		ProdAER_1T_realtime := (INT_TO_REAL(ProducaoProgramada_AER_1T) / (MinDispAER_1T)) * ((
		(INT_TO_REAL(hora)-INT_TO_REAL(HoraInicio1Turno))*60)-INT_TO_REAL(MinInicio1Turno) + INT_TO_REAL(minuto)-10-20-15);
	
		EficAER_1T_realtime := ( INT_TO_REAL(CNT_PRD_AER_1T) / ProdAER_1T_realtime ) * 100;
		END_IF
		
				IF hora > 12 AND hora < 15 AND minuto < 9 THEN

		ProdAER_1T_realtime := (INT_TO_REAL(ProducaoProgramada_AER_1T) / (MinDispAER_1T)) * ((
		(INT_TO_REAL(hora)-INT_TO_REAL(HoraInicio1Turno))*60)-INT_TO_REAL(MinInicio1Turno) + INT_TO_REAL(minuto)-10-20-15-60-10);
	
		EficAER_1T_realtime := ( INT_TO_REAL(CNT_PRD_AER_1T) / ProdAER_1T_realtime ) * 100;
		END_IF
//HABILITA RTC==========================
	IF xEnable = TRUE THEN
	Result := GetDateAndTime(DATEANDTIME);
	END_IF
//HABILITA RTC==========================

//==============Habilita contadores 1º turno ================
IF (hora = HoraInicio1Turno AND minuto = MinInicio1Turno)  THEN
HabContAER_1T := TRUE;
HabContAER_3T := FALSE;
END_IF 


//==============Contador e Eficiencia AER 1 TURNO de cartuchos==========
IF HabContAER_1T = TRUE THEN 
PULSO_CNT_AER_1T(CLK:=CNT_AER);	
		IF PULSO_CNT_AER_1T.Q = TRUE THEN
		CNT_PRD_AER_1T := CNT_PRD_AER_1T+1;	
		END_IF
END_IF
EficienciaAER_1T := (INT_TO_REAL(CNT_PRD_AER_1T) / INT_TO_REAL(ProducaoProgramada_AER_1T) ) * 100;

//=====================1º TURNO ========================

//=====================2º TURNO ========================

	//10 minutos - Reunião / DSS / Treinamento
	//20 minutosPartida de linha / Parada de Linha
	//15 minutosRefeições (Café / Almoço / Janta)
	//60 minutosRefeições (Café / Almoço / Janta)
	//10 minutosPartida de linha / Parada de Linha
	IF hora = 0 THEN 
		hora := 24;
	END_IF
	
		MinDispAER_2T := (((INT_TO_REAL (HoraFim2Turno) - INT_TO_REAL(HoraInicio2Turno) )*60)-
		INT_TO_REAL(MinInicio2Turno)+INT_TO_REAL(MinFim2Turno)-10-20-15-60-10);
		
	IF (hora > 15 AND minuto > 8) AND hora < 17 THEN

		ProdAER_2T_realtime := (INT_TO_REAL(ProducaoProgramada_AER_2T) / (MinDispAER_2T)) * ((
		(INT_TO_REAL(hora)-INT_TO_REAL(HoraInicio2Turno))*60)-INT_TO_REAL(MinInicio2Turno) + INT_TO_REAL(minuto)-10-20);
	
		EficAER_2T_realtime := ( INT_TO_REAL(CNT_PRD_AER_2T) / ProdAER_2T_realtime ) * 100;
		END_IF
		
			IF hora > 17 AND hora < 20 THEN

		ProdAER_2T_realtime := (INT_TO_REAL(ProducaoProgramada_AER_2T) / (MinDispAER_2T)) * ((
		(INT_TO_REAL(hora)-INT_TO_REAL(HoraInicio2Turno))*60)-INT_TO_REAL(MinInicio2Turno) + INT_TO_REAL(minuto)-10-20-15);
	
		EficAER_2T_realtime := ( INT_TO_REAL(CNT_PRD_AER_2T) / ProdAER_2T_realtime ) * 100;
		END_IF
		
				IF hora > 20 AND hora < 24 THEN

		ProdAER_2T_realtime := (INT_TO_REAL(ProducaoProgramada_AER_2T) / (MinDispAER_2T)) * ((
		(INT_TO_REAL(hora)-INT_TO_REAL(HoraInicio2Turno))*60)-INT_TO_REAL(MinInicio2Turno) + INT_TO_REAL(minuto)-10-20-15-60-10);
	
		EficAER_2T_realtime := ( INT_TO_REAL(CNT_PRD_AER_2T) / ProdAER_2T_realtime ) * 100;
		END_IF
//==============Contador e Eficiencia AER 2 TURNO de cartuchos==========
//==============Habilita contadores 2º turno ================
IF (hora = HoraInicio2Turno AND minuto = MinInicio2Turno)  THEN
HabContAER_2T := TRUE;
HabContAER_1T := FALSE;
END_IF 
IF HabContAER_2T = TRUE THEN 
PULSO_CNT_AER_2T(CLK:=CNT_AER);	
		IF PULSO_CNT_AER_2T.Q = TRUE THEN
		CNT_PRD_AER_2T := CNT_PRD_AER_2T+1;	
		END_IF
END_IF
EficienciaAER_2T := (INT_TO_REAL (CNT_PRD_AER_2T) / INT_TO_REAL (ProducaoProgramada_AER_2T)  ) * 100;

//=====================2º TURNO ========================

//=====================3º TURNO ========================
//==============Contador e Eficiencia AER 3 TURNO de cartuchos==========

//==============Habilita contadores 3º turno ================
//10 minutos - Reunião / DSS / Treinamento
	//20 minutosPartida de linha / Parada de Linha
	//15 minutosRefeições (Café / Almoço / Janta)
	//60 minutosRefeições (Café / Almoço / Janta)
	//10 minutosPartida de linha / Parada de Linha
	IF hora = 0 THEN 
		hora := 24;
	END_IF
	
		MinDispAER_3T := (((INT_TO_REAL (HoraFim3Turno) - INT_TO_REAL(HoraInicio3Turno) )*60)-
		INT_TO_REAL(MinInicio3Turno)+INT_TO_REAL(MinFim3Turno)-10-20-15-60-10);
		
	IF ((hora > 0 OR hora = 24) AND minuto > 32) AND hora < 02 THEN

		ProdAER_3T_realtime := (INT_TO_REAL(ProducaoProgramada_AER_3T) / (MinDispAER_3T)) * ((
		(INT_TO_REAL(hora)-INT_TO_REAL(HoraInicio3Turno))*60)-INT_TO_REAL(MinInicio3Turno) + INT_TO_REAL(minuto)-10-20);
	
		EficAER_3T_realtime := ( INT_TO_REAL(CNT_PRD_AER_3T) / ProdAER_3T_realtime ) * 100;
		END_IF
		
			IF hora > 17 AND hora < 20 THEN

		ProdAER_3T_realtime := (INT_TO_REAL(ProducaoProgramada_AER_3T) / (MinDispAER_3T)) * ((
		(INT_TO_REAL(hora)-INT_TO_REAL(HoraInicio3Turno))*60)-INT_TO_REAL(MinInicio3Turno) + INT_TO_REAL(minuto)-10-20-15);
	
		EficAER_3T_realtime := ( INT_TO_REAL(CNT_PRD_AER_3T) / ProdAER_3T_realtime ) * 100;
		END_IF
		
				IF hora > 20 AND hora < 24 THEN

		ProdAER_3T_realtime := (INT_TO_REAL(ProducaoProgramada_AER_3T) / (MinDispAER_3T)) * ((
		(INT_TO_REAL(hora)-INT_TO_REAL(HoraInicio3Turno))*60)-INT_TO_REAL(MinInicio3Turno) + INT_TO_REAL(minuto)-10-20-15-60-10);
	
		EficAER_3T_realtime := ( INT_TO_REAL(CNT_PRD_AER_3T) / ProdAER_3T_realtime ) * 100;
		END_IF
//==============Contador e Eficiencia AER 3 TURNO de cartuchos==========
//==============Habilita contadores 3º turno ================
IF (hora = HoraInicio3Turno AND minuto = MinInicio3Turno)  THEN
HabContAER_3T := TRUE;
HabContAER_2T := FALSE;
END_IF 
IF HabContAER_3T = TRUE THEN 
PULSO_CNT_AER_3T(CLK:=CNT_AER);	
		IF PULSO_CNT_AER_3T.Q = TRUE THEN
		CNT_PRD_AER_3T := CNT_PRD_AER_3T+1;	
		END_IF
END_IF
EficienciaAER_3T := (INT_TO_REAL (CNT_PRD_AER_3T) / INT_TO_REAL (ProducaoProgramada_AER_3T)  ) * 100;


IF (hora = HoraInicio3Turno AND minuto = MinInicio3Turno)  THEN
HabContAER_3T := TRUE;
HabContAER_2T := FALSE;
END_IF 
IF HabContAER_3T = TRUE THEN 
PULSO_CNT_AER_3T(CLK:=CNT_AER);	
		IF PULSO_CNT_AER_3T.Q = TRUE THEN
		CNT_PRD_AER_3T := CNT_PRD_AER_3T+1;	
		END_IF
END_IF
EficienciaAER_3T := (INT_TO_REAL (CNT_PRD_AER_3T) / INT_TO_REAL(ProducaoProgramada_AER_3T)  ) * 100;
//=====================3º TURNO ========================

END_PROGRAM

// Device/Application/ampliacao_transferencia
PROGRAM ampliacao_transferencia

VAR
	BA_03_INV : INV_MODBUS;
	BB_02_INV : INV_MODBUS;
	MH_01_INV : INV_MODBUS;
	MH_02_INV : INV_MODBUS;
	
	AUX_BA_03_HAB : BOOL;
	AUX_BB_02_HAB : BOOL;
	AUX_MH_01_HAB : BOOL;
	AUX_MH_02_HAB : BOOL;
	AUX_BA_03_PRESET: REAL;
	CTRL_BB2 : PD;
	BB_02_PRT_MAN : BOOL;
	AUX_BA_03_FLT_PRESS : BOOL;
	
	AUX_BB2_PRST_VEL : REAL;
	
	
	R_BB_02_REF_VEL : REAL;
	R_PRST_PRESS_BB : REAL;
	R_BB_02_PRS_VEL : REAL;
	
	
	TMR_FALHA_PRESSAO_BBALTA3_ALARME : TON;
END_VAR


(* PARAMENTROS DO INVERSOR DA BOMBA DE ALTA PRESSÃO 03*)
BA_03_INV (
	LIGA := BA_03_CMDS,
	CMD_RESET := BTS_RSTAL,
	CMD_STOP := AL_GERAL,
	CMD_HAB := AUX_BA_03_HAB,
	REF_VEL := BA_03_REF_VEL,
	STATUS := BA_03_ST,
	FALHA := BA_03_FLT,
	PRESET := AUX_BA_03_PRESET,
	LIGADO => BA_03_CMD,
	HABILITADO => BA_03_HAB,
	STOP => BA_03_STP,
	RESET => BA_03_RST,
	VEL => BA_03_ST_VELS,
	STS_INV => BA_03_STS,
	FLT_INV => BA_03_FLTS,
	PRT_VEL => BA_03_PRS_VEL);
	
	
	(* PARAMENTROS DO INVERSOR DA BOMBA DE BAIXA PRESSÃO 02*)
BB_02_INV (
	LIGA := BB_02_CMDS,
	CMD_RESET := BTS_RSTAL,
	CMD_STOP := AL_GERAL,
	CMD_HAB := AUX_BB_02_HAB,
	//REF_VEL := 
	STATUS := BB_02_ST,
	FALHA := BB_02_FLT,
	PRESET := AUX_BB2_PRST_VEL,
	LIGADO => BB_02_CMD,
	HABILITADO => BB_02_HAB,
	STOP => BB_02_STP,
	RESET => BB_02_RST,
	//VEL => 
	STS_INV => BB_02_STS,
	FLT_INV => BB_02_FLTS,
	PRT_VEL => BB_02_PRS_VEL);
	
		(* PARAMENTROS DO INVERSOR DO MOINHO 01*)
MH_01_INV (
	LIGA := MH_01_CMDS,
	CMD_RESET := BTS_RSTAL,
	CMD_STOP := AL_GERAL,
	CMD_HAB := AUX_MH_01_HAB,
	//REF_VEL := 
	STATUS := MH_01_ST,
	FALHA := MH_01_FLT,
	//PRESET := 
	LIGADO => MH_01_CMD,
	HABILITADO => MH_01_HAB,
	STOP => MH_01_STP,
	RESET => MH_01_RST,
	//VEL => 
	STS_INV => MH_01_STS,
	FLT_INV => MH_01_FLTS,
	//PRT_VEL => 
);

	(* PARAMENTROS DO INVERSOR DO MOINHO 01*)
MH_02_INV (
	LIGA := MH_02_CMDS,
	CMD_RESET := BTS_RSTAL,
	CMD_STOP := AL_GERAL,
	CMD_HAB := AUX_MH_02_HAB,
	//REF_VEL := 
	STATUS := MH_02_ST,
	FALHA := MH_02_FLT,
	//PRESET := 
	LIGADO => MH_02_CMD,
	HABILITADO => MH_02_HAB,
	STOP => MH_02_STP,
	RESET => MH_02_RST,
	//VEL => 
	STS_INV => MH_02_STS,
	FLT_INV => MH_02_FLTS,
	//PRT_VEL => 
);

                   (*LOGICA DA BOMBA DE ALTA 03*)
//----------------------------------------------------------------------------------

//COMANDO LIGA DA BOMBA DE ALTA 03				   
IF  (SD_BB=TRUE OR BB_02_ST = TRUE) AND  PRESSAO_ALTA_LINHA_ALTA = FALSE THEN
IF (NOT SD_BA1) OR (NOT SD_BA2) THEN
	AUX_BA_03_HAB := TRUE;
	END_IF
END_IF

//SETPOINT VELOCIDADE DE BOMBA DE ALTA 03
IF BA_03_ST THEN
	AUX_BA_03_PRESET := PRST_VEL_BA1;
	ELSE 
		AUX_BA_03_PRESET := 0;
	END_IF

                   (*LOGICA DA BOMBA DE BAIXA 02*)
//----------------------------------------------------------------------------------

// COMANDO LLIGA DA BOMBA DE BAIXA 02
	IF SD_BB = FALSE AND NIVEL_MINIMO_MXE = FALSE AND PRESSAO_ALTA_LINHA_ALTA = FALSE THEN
	AUX_BB_02_HAB := TRUE;
	ELSE
	AUX_BB_02_HAB := FALSE;
END_IF
	//move velocidade da bomba de baixa 02 em manual
 IF (BB_02_ST = TRUE AND BB_AUTOM = FALSE) THEN
		AUX_BB2_PRST_VEL := BB_02_PRS_VEL;
	
END_IF
		
	
	// SETPIOINT VAI A ZERO SE NAO ESTIVER FUNCIONANDO
IF BB_02_ST = FALSE THEN 
	AUX_BB2_PRST_VEL := 0;
	END_IF
	
		//move velocidade da bomba de baixa 02 em automatico (AMPLIAÇÃO)
	IF (BB_02_ST = TRUE AND BB_AUTOM = TRUE) THEN
	AUX_BB2_PRST_VEL := (REAL_TO_WORD (PRESSAO_BOMBA));
	END_IF
	

	
	(* CONTROLE PID DA BOMBA DE BAIXA PRESSÃO 02
//VERIFICAR SE É NECESSARIO CONVERTER OS VALORES DO PID EM REAL SO 
IF BB_02_ST = TRUE THEN
	CTRL_BB2 (
		ACTUAL:= R_BB_02_REF_VEL,
		SET_POINT := R_PRST_PRESS_BB,
		KP := 1,
		TV := 0.5,
		Y_MANUAL := R_BB_02_PRS_VEL,
		Y_MIN := 0,
		Y_MAX := 100, // AJUSTAR VALORES LIMITES
		MANUAL := BB_02_PRT_MAN,
		RESET := AUX_BB_02_HAB,
		Y => R_PRESSAO_BOMBA);
	END_IF *)
		
// comando dos moinho (com intertravamento entre eles	
	IF MH_01_ST THEN
			AUX_MH_02_HAB := FALSE;
		ELSE
			AUX_MH_02_HAB := TRUE;
		END_IF
		
		IF MH_02_ST THEN
			AUX_MH_01_HAB := FALSE;
		ELSE
			AUX_MH_01_HAB := TRUE;
		END_IF
		
		
		//Falha de pressão Bomba alta 3
IF BA_03_ST = TRUE AND BA_03_PRESS = TRUE THEN
	AUX_BA_03_FLT_PRESS:=TRUE;
ELSE
	AUX_BA_03_FLT_PRESS:= FALSE;
END_IF

TMR_FALHA_PRESSAO_BBALTA3_ALARME(IN:=AUX_BA_03_FLT_PRESS, PT:=T#15S);

IF TMR_FALHA_PRESSAO_BBALTA3_ALARME.Q = TRUE THEN
	BA_03_FLT_PRESS :=TRUE;
END_IF

END_PROGRAM

// Device/Application/inv_modbus
FUNCTION_BLOCK inv_modbus

VAR_INPUT
	LIGA : BOOL; // SINAL DO COMANDO DE LIGA\DESLIGA
	CMD_RESET : BOOL; // SINAL DE COMANDO DE RESET
	CMD_STOP : BOOL; // SINAL DO BOTÃO DE EMERGENCIA
	CMD_HAB : BOOL; //SINAL DE HABILITAÇÃO DO INVERSOR
	REF_VEL : DWORD; // REFERENCIA DE VELOCIDADE
	STATUS : BOOL; // STATUS DO INVERSOR 
	FALHA : BOOL; // SINAL DE FALHA DO INVERSOR
	PRESET : REAL; // PRESET DE VELOCIDADE
		
END_VAR
VAR_OUTPUT
	LIGADO : BOOL; //COMANDO LIGADO
	HABILITADO : BOOL; // INVERSOR HABILITADO
	STOP : BOOL; //EMERGENCIA ATUADA
	RESET : BOOL; //COMANDO RESET
	VEL : WORD; //SET DE VELOCIDADE
	STS_INV : BOOL; //STATUS DO INVERSOR
	FLT_INV : BOOL; //INVERSOR EM FALHA
	PRT_VEL : WORD; // PRESET
		
END_VAR

IF LIGA AND STOP AND CMD_HAB AND NOT FALHA THEN
IF LIGADO := FALSE THEN
LIGADO := TRUE;
ELSE
	LIGADO := FALSE;
END_IF
ELSE 
	LIGADO := FALSE;
	
END_IF

IF CMD_HAB AND STOP AND NOT FALHA THEN
HABILITADO := TRUE;
ELSE
	HABILITADO := FALSE;
END_IF

	
	

RESET := CMD_RESET;
STOP := CMD_STOP;
STS_INV := STATUS;
FLT_INV := FALHA;
PRT_VEL := (REAL_TO_WORD (PRESET));
VEL  := ( DWORD_TO_WORD (REF_VEL));

END_FUNCTION_BLOCK
